Staubli VAL3: Main.pjx

--- Main.pjx ---
Parameters version=s7.3 stackSize=5000 millimeterUnit=true
Program file=SIMPLE_MSG.pgx
Program file=TASK_MANAGER.pgx
Program file=consume.pgx
Program file=consumeAny.pgx
Program file=start.pgx
Program file=stop.pgx
Data file=Main.dtx
Library alias=trajMsg path=Disk://JointTrajPtFull/JointTrajPtFull.pjx autoload=true password=
Library alias=msgSpec path=Disk://SimpleMessage/SimpleMessage.pjx autoload=true password=

--- Main.dtx ---
bool bInputBuffering
bool bTaskManager
jointRx jHome
mdesc mNomSpeed
num nInputBuffer[136]
  [0] = 1
  [4] = 255
  [5] = 255
  [6] = 255
  [7] = 255
  [8] = 15
  [14] = 164
  [15] = 66
  [58] = 72
  [59] = 66
  [98] = 200
  [99] = 65
  [102] = 200
  [103] = 65
num nMessageBuffer[34 4]
  [0,0] = 1
  [1,0] = 255
  [1,1] = 255
  [1,2] = 255
  [1,3] = 255
  [2,0] = 15
  [3,2] = 164
  [3,3] = 66
  [14,2] = 72
  [14,3] = 66
  [24,2] = 200
  [24,3] = 65
  [25,2] = 200
  [25,3] = 65
sio siConn = {link=Socket\subscriber}
sio soConn = {link=Socket\publisher}
string sInputBuffering = "subscriber"

--- start.pgx ---
program start()
  local num l_nSioCtrl
begin
  bInputBuffering=true
  sInputBuffering="subscriber"
  bTaskManager=true
  cls()
  resetMotion()
  userPage()
  l_nSioCtrl=sioCtrl(siConn,"timeout",5)
  if (l_nSioCtrl<0)
    putln("Could not set the timeout")
  endIf
  putln("Starting task")
  l_nSioCtrl=sioCtrl(soConn,"timeout",5)
  if (l_nSioCtrl<0)
    putln("Could not set the timeout")
  endIf
  taskCreate sInputBuffering,50,SIMPLE_MSG(trajMsg:prefix.nLength,trajMsg:header.nMsgType)
  taskCreate "t_manage",10,TASK_MANAGER()
end

--- consume.pgx ---
program consume(num& x_nStatus (dimensions=1), num x_nReference (dimensions=1))
  local num l_nConnStatus
  local num l_nData[4]
  local num l_nValue
  local num l_nBinaryStatus
begin
  // consumes 4 bytes and verifes with the reference
  // does nothing if first return parameter is not 0
  // return
  //    -2 - timeout
  //    -1 - unexpected value
  //     0 - expected value
  if x_nStatus<0
    return
  endIf
  x_nStatus=-1
  l_nConnStatus=sioGet(siConn,l_nData)
  if l_nConnStatus==4
    l_nBinaryStatus=fromBinary(l_nData,4,"4l",l_nValue)
    if l_nData==x_nReference and l_nBinaryStatus==1
      x_nStatus=0
    endIf
  elseIf l_nConnStatus==-1
    x_nStatus=-2
  endIf
end

--- consumeAny.pgx ---
program consumeAny(num& x_nStatus (dimensions=1))
  local num l_nData[4]
begin
  // consumes 4 bytes and verifes with the reference
  // does nothing if first return parameter is not 0
  // return
  //    -2 - timeout
  //    -1 - unsuccessful
  //     0 - successfuly received (consumed) 4 bytes
  if x_nStatus<0
    return
  endIf
  x_nStatus=sioGet(siConn,l_nData)
  if x_nStatus==4
    x_nStatus=0
  elseIf x_nStatus==-1
    x_nStatus=-2
  else
    x_nStatus=-1
  endIf
end

--- SIMPLE_MSG.pgx ---
program SIMPLE_MSG(num x_nLength, num x_nMsgType)
  local num l_nStatus
  local num l_nBytesToGet
  local num i
  local num j
  local num k
  local num l_nRespBuffer[152]
  local joint l_jJoint
  local mdesc l_mMdesc
begin
  // This TASK specialises in receiving ros simple messages
  // thus it validates prefix and the header and then accepts
  // the bytes from the body
  // payload length in bytes minus header size (12 bytes)
  l_nBytesToGet=x_nLength-12
  resize(nInputBuffer,1,l_nBytesToGet)
  resize(nMessageBuffer,1,l_nBytesToGet/4)
  resize(nMessageBuffer,2,4)
  while (bInputBuffering)
    l_nStatus=0
    // prefix
    call consume(l_nStatus,x_nLength)
    // header
    call consume(l_nStatus,x_nMsgType)
    call consume(l_nStatus,msgSpec:commType.nRequest)
    call consumeAny(l_nStatus)
    if l_nStatus<0
      if l_nStatus==-2
        putln("Timeout.")
      else
        putln("Bad request header/prefix.")
      endIf
    else
      // get the body
      j=0
      k=0
      while j<l_nBytesToGet/4
        l_nStatus=sioGet(siConn,nInputBuffer)
        if l_nStatus>0
          for i=0 to l_nStatus-1
            nMessageBuffer[j,k]=nInputBuffer[i]
            k=k+1
            if k>3
              k=0
              j=j+1
            endIf
          endFor
        endIf
      endWhile
      // decode the body
      call trajMsg:decode(l_nStatus,nMessageBuffer)
      delay(0)
      // modify the header for acknowledge message
      trajMsg:header.nCommType=msgSpec:commType.nResponse
      if l_nStatus<0
        trajMsg:header.nReplyCode=msgSpec:replyType.nFailure
        putln("Failed to decode the body of the message.")
      else
        trajMsg:header.nReplyCode=msgSpec:replyType.nSuccess
      endIf
      // encode the acknowledge message
      call trajMsg:encode(l_nStatus,l_nRespBuffer)
      if l_nStatus<0
        putln("Failed to encode the acknowledge message.")
        trajMsg:header.nReplyCode=msgSpec:replyType.nFailure
      endIf
      // send the acknowledge message
      l_nStatus=sioSet(soConn,l_nRespBuffer)
      if l_nStatus<0
        putln("Failed to send acknowledge response: "+toString("",l_nStatus))
      else
        // convert the message to joint & motion descirptor
        call trajMsg:convert(l_jJoint,l_mMdesc)
        // print the joint values
        put(toString("5",l_jJoint.j1)+","+toString("5",l_jJoint.j2)+","+toString("5",l_jJoint.j3))
        putln(","+toString("5",l_jJoint.j4)+","+toString("5",l_jJoint.j5)+","+toString("5",l_jJoint.j6))
        // apply the point to flange and add it to the motion queue
        movej(l_jJoint,flange,l_mMdesc)
      endIf
    endIf
  endWhile
end

--- stop.pgx ---
program stop()
  local num l_nI
begin
  putln("TaskStatus: "+toString("",taskStatus(sInputBuffering)))
  bInputBuffering=false
  bTaskManager=false
  resetMotion()
  //wait(taskStatus(sInputBuffering)==0)
  delay(2)
  if taskStatus(sInputBuffering)!=0
    taskKill(sInputBuffering)
  endIf
  putln("TaskStatus: "+toString("",taskStatus(sInputBuffering)))
  putln("Stopped.")
end

--- TASK_MANAGER.pgx ---
program TASK_MANAGER()
begin
  while (bTaskManager)
    if taskStatus(sInputBuffering)==150
      taskKill(sInputBuffering)
      resetMotion()
      putln("Restart SIMPLE_MSG task.")
      taskCreate sInputBuffering,50,SIMPLE_MSG(trajMsg:prefix.nLength,trajMsg:header.nMsgType)
    endIf
  endWhile
end
